// TIA Portal project "Automatisierte_Nullfüllstation_FUP" (V16)

(* hardware
DEVICE "S7-1200 station_1"  S7-1200 Station
   slot 0: "Rack_0"  S7-1200 Rack  Rack  V1.0
   slot 1: "PLC_1"  CPU 1212C DC/DC/DC  6ES7 212-1AE40-0XB0  V4.4
*)

// ===== PLC "PLC_1"  CPU 1212C DC/DC/DC =====

VAR_GLOBAL   // PLC tag table "Default tag table"
   "Eingang_Näherungssensor" AT %I0.0 : Bool;
   "Eingang_Ultraschallfüllstandsensor" AT %I0.1 : Bool;
   "Kontaktstelle Farbsensor (ROT)" AT %I0.2 : Bool;
   "Kontaktstelle Farbsensor (BLAU)" AT %I0.3 : Bool;
   "Ausgang_Motor" AT %Q0.0 : Bool;
   "Ausgang_Walnusszufuhrklappe" AT %Q0.1 : Bool;
   "Ausgang_Pekanzufuhrklappe" AT %Q0.2 : Bool;
   "Näherungssensor_Bit" AT %M0.0 : Bool;
   "Ultraschallfüllstandsensor_Bit" AT %M0.1 : Bool;
   "Farbsensor (ROT)_Bit" AT %M0.2 : Bool;
   "Farbsensor (BLAU)_Bit" AT %M0.3 : Bool;
   "Motor_Bit" AT %M0.4 : Bool;
   "Walnusszufuhrklappe_Bit" AT %M0.5 : Bool;
   "Pekanzufuhrklappe_Bit" AT %M0.6 : Bool;
   "Modus" AT %MW2 : Int;
END_VAR

DATA_BLOCK "IO_DB"   // DB1
{ S7_Optimized_Access := 'TRUE' }
VERSION : 0.1
// stored: InstanceOfName IO
"IO"
BEGIN
END_DATA_BLOCK

DATA_BLOCK "Steuerlogik_DB"   // DB2
{ S7_Optimized_Access := 'TRUE' }
VERSION : 0.1
// stored: InstanceOfName Steuerlogik
"Steuerlogik"
BEGIN
END_DATA_BLOCK

FUNCTION_BLOCK "IO"   // FB1, FBD
{ S7_Optimized_Access := 'TRUE' }
VERSION : 0.1
BEGIN

REGION Network 1
   // Eingänge
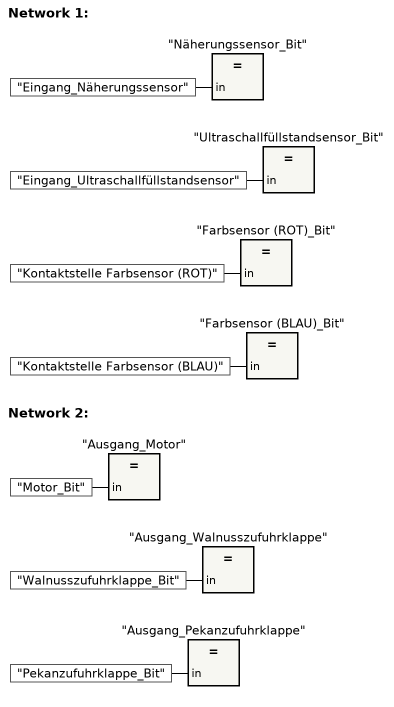
   "Näherungssensor_Bit" := "Eingang_Näherungssensor";
   "Ultraschallfüllstandsensor_Bit" := "Eingang_Ultraschallfüllstandsensor";
   "Farbsensor (ROT)_Bit" := "Kontaktstelle Farbsensor (ROT)";
   "Farbsensor (BLAU)_Bit" := "Kontaktstelle Farbsensor (BLAU)";
END_REGION

REGION Network 2
   // Ausgänge
   "Ausgang_Motor" := "Motor_Bit";
   "Ausgang_Walnusszufuhrklappe" := "Walnusszufuhrklappe_Bit";
   "Ausgang_Pekanzufuhrklappe" := "Pekanzufuhrklappe_Bit";
END_REGION
END_FUNCTION_BLOCK

FUNCTION_BLOCK "Steuerlogik"   // FB2, FBD
{ S7_Optimized_Access := 'TRUE' }
VERSION : 0.1
// Modus:
// 1 = Motor an 
// 2 = Füllmodus
BEGIN

REGION Network 1
   // Steuerlogik für Motor
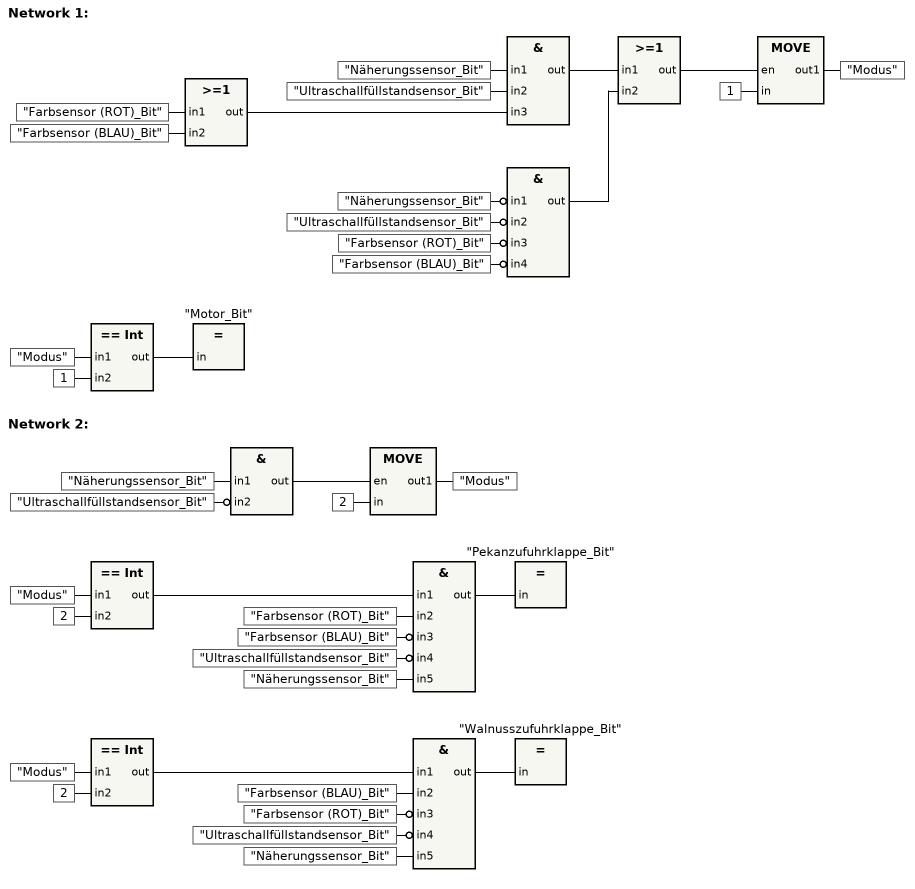
   IF ("Näherungssensor_Bit" AND "Ultraschallfüllstandsensor_Bit" AND ("Farbsensor (ROT)_Bit" OR "Farbsensor (BLAU)_Bit")) OR (NOT "Näherungssensor_Bit" AND NOT "Ultraschallfüllstandsensor_Bit" AND NOT "Farbsensor (ROT)_Bit" AND NOT "Farbsensor (BLAU)_Bit") THEN
       "Modus" := 1;
   END_IF;
   "Motor_Bit" := "Modus" = 1;
END_REGION

REGION Network 2
   // Steuerlogik beim Füllmodus
   IF "Näherungssensor_Bit" AND NOT "Ultraschallfüllstandsensor_Bit" THEN "Modus" := 2; END_IF;
   "Pekanzufuhrklappe_Bit" := ("Modus" = 2) AND "Farbsensor (ROT)_Bit" AND NOT "Farbsensor (BLAU)_Bit" AND NOT "Ultraschallfüllstandsensor_Bit" AND "Näherungssensor_Bit";
   "Walnusszufuhrklappe_Bit" := ("Modus" = 2) AND "Farbsensor (BLAU)_Bit" AND NOT "Farbsensor (ROT)_Bit" AND NOT "Ultraschallfüllstandsensor_Bit" AND "Näherungssensor_Bit";
END_REGION
END_FUNCTION_BLOCK

ORGANIZATION_BLOCK "Main"   // OB1, LAD, ProgramCycle
TITLE = "Main Program Sweep (Cycle)"
{ S7_Optimized_Access := 'TRUE' }
VERSION : 0.1
// PROJEKTBESCHREIBUNG.: In diesem Projekt geht um die automatische Nussabfüllmaschine. Die Anlage besteht aus einem Motor, einem Förderband, einem Näherungssensor, zwei Nusstrichter (Pekan- und Walnusstrichter) mti Zufuhrklappen, einem Farbsensor (erkennt rot und blau) und einem Ultraschallfüllstandsensor. Die Reihenfolge der Steuerlogik ist wie folgt:
// 1)  Auf dem Förderband liegen die abzufüllenden Kartonverpackungen. Der Motor geht an und somit bewegt den Förderband bis der Näherungssensor die Kartonverpackung erkennt.
// 2) Auf der Kartonverpackung ist jeweils eine rote oder blaue Etikettierung.Der Farbsensor erkennt die Farbe und anhand dieser Farbe (rot für Pekannüsse und blau für Walnüsse) wird jeweiligen Zufuhrklappen zur Befüllung geöffnet.
// 3) Der Ultraschallfüllstandsensor misst ständig ,ob die Verpackung voll ist. Falls ja, die Zufuhrklappe ist geschlossen und der Förderband bewegt die befüllte Verpackung weiter.  
// 
// TESTKRITERIEN:
// 1)Um zu beginnen, starten Sie Ihr Programm auf PLCSIM. Der Fördermotor sollte sofort anlaufen, aber beide Trichter sollten ausgeschaltet sein.
// 
// 2)Als Nächstes erzwingen Sie nur den Näherungsschalter (geschlossen). Der Fördermotor sollte sich abschalten, und beide Trichter sollten ausgeschaltet bleiben.
// 
// 3)Drittens lassen Sie den Näherungsschalter geschlossen und erzwingen zusätzlich die rote Lichtschranke. Der Fördermotor und der Walnuss-Trichter sollten ausgeschaltet bleiben, aber der Pekannuss-Trichter sollte einschalten.
// 
// 4)Viertens lassen Sie den Näherungsschalter geschlossen, schalten die rote Lichtschranke aus und erzwingen die blaue Lichtschranke. Der Fördermotor sollte ausgeschaltet bleiben, der Pekannuss-Trichter sollte ausgehen und der Walnuss-Trichter sollte einschalten.
// 
// 5)Als Nächstes erzwingen Sie den Füllstandsschalter. Beide Trichter sollten ausgeschaltet werden und der Förderer sollte wieder anlaufen, um die Kiste weiterzubewegen.
// 
// 6)Zum Schluss schalten Sie den Näherungsschalter, den Füllstandsschalter und beide Lichtschranken aus. Beide Trichter sollten ausgeschaltet bleiben und der Förderer sollte weiterlaufen.
// 7)
// Zusatztest: Bei geöffnetem Näherungsschalter und Füllstandsschalter erzwingen Sie beide Lichtschranken. Keiner der Trichter sollte einschalten. (Wir wollen kein Produkt freigeben, wenn keine Kiste zum Auffangen da ist.)
   VAR_INPUT
      Initial_Call : Bool;   // Initial call of this OB
      Remanence : Bool;   // =True, if remanent data are available
   END_VAR
BEGIN

REGION Network 1
   // IO
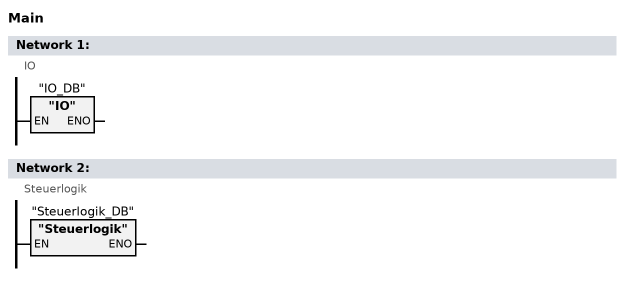
   RUNG wire#powerrail
      "IO_DB"()
   END_RUNG
   // the same network as SCL:
   "IO_DB"();   // "IO"
END_REGION

REGION Network 2
   // Steuerlogik
   RUNG wire#powerrail
      "Steuerlogik_DB"()
   END_RUNG
   // the same network as SCL:
   "Steuerlogik_DB"();   // "Steuerlogik"
END_REGION
END_ORGANIZATION_BLOCK